Staubli VAL3: tRobot.pgx

program tRobot()
begin
  resetMotion(jStart)

  while true
    movej(appro(pPick,trAppro),flange,mNomSpeed)
    movel(pPick,flange,mNomSpeed)
    waitEndMove()
    movel(appro(pPick,trAppro),flange,mNomSpeed)

    movej(appro(pPlace,trAppro),flange,mNomSpeed)
    movel(pPlace,flange,mNomSpeed)
    waitEndMove()
    movel(appro(pPlace,trAppro),flange,mNomSpeed)

    delay(0)
  endWhile
end
